// TwinCAT 3 PLC project Project_02
// ProgramVersion: 3.1.4024.0
// libraries:
//   Tc2_Standard, * (Beckhoff Automation GmbH)
//   Tc2_System, * (Beckhoff Automation GmbH)
//   Tc3_Module, * (Beckhoff Automation GmbH)
// project tree:
//   DUTs/ DUT.TcTLEO
//   GVLs/ InputOutput.TcGVL
//   / PlcTask.TcTTO
//   POUs/ FB_MSF.TcPOU, FB_oscillatore.TcPOU, MAIN.TcPOU

CONFIGURATION Project_02
    RESOURCE PLC ON TwinCAT3
        TASK PlcTask(INTERVAL := T#10ms, PRIORITY := 20);
        PROGRAM MAIN WITH PlcTask : MAIN;
    END_RESOURCE
END_CONFIGURATION

// ---- DUTs/DUT.TcTLEO
{attribute 'qualified_only'}
{attribute 'strict'}

TYPE STATI :
(
	S0 := 0, S1, S2, S3, SE, SA
);
END_TYPE

// ---- GVLs/InputOutput.TcGVL
{attribute 'qualified_only'}
VAR_GLOBAL
	start  : BOOL;
	stop   : BOOL;
	emg    : BOOL;
	ack    : BOOL;
	fc1    : BOOL;
	fc2    : BOOL;
	
	H1     : BOOL;
	HEMG   : BOOL;
	M      : BOOL;
	libero : BOOL;
	
END_VAR

// ---- POUs/MAIN.TcPOU
PROGRAM MAIN
VAR
	nastro: FB_MSF();
	emg: BOOL;
END_VAR


nastro(
	start:= InputOutput.start, 
	stop:= InputOutput.stop, 
	emg:= InputOutput.emg, 
	ack:= InputOutput.ack, 
	fc1:= InputOutput.fc1, 
	fc2:= InputOutput.fc2, 
	H1=> InputOutput.H1, 
	HEMG=> InputOutput.HEMG, 
	M=> InputOutput.M, 
	libero=> InputOutput.libero);

END_PROGRAM

// ---- POUs/FB_MSF.TcPOU
FUNCTION_BLOCK FB_MSF
VAR_INPUT
	start: BOOL;
	stop : BOOL := TRUE;
	emg  : BOOL := TRUE;
	ack  : BOOL;
	fc1  : BOOL;
	fc2  : BOOL;
END_VAR
VAR_OUTPUT
	H1   : BOOL;
	HEMG : BOOL;
	M    : BOOL;
	// il nastro è libero
	libero : BOOL;
END_VAR
VAR
	
	// abilitazione dell’automatismo
	enable : BOOL := TRUE;
	// condizioni di transizione
	tr_S0_S1 : BOOL;
	tr_S1_S2 : BOOL;
	tr_S2_S3 : BOOL;
	tr_S3_S1 : BOOL;
	tr_S3_S0 : BOOL;
	tr_SE_SA : BOOL;
	tr_SA_S0 : BOOL;
	// variabile di stato
	stato : STATI := STATI.S0;
	// timers
	T31 : TON();
	TA0 : TON();
	// triggers per segnalazione nastro libero
	pckin : R_TRIG();
	pckout: R_TRIG();
	// lampeggio
	osc : FB_oscillatore();	
END_VAR

(*
1.aggiornamento delle condizioni di abilitazione (stop, allarmi, etc)
2.aggiornamento di timers, contatori, triggers sui fronti
3.valutazione della condizione di arresto nominale
4.valutazione della condizione di arresto di emergenza
5.aggiornamento delle condizioni di transizione di stato
6.switch-case della MSF
7.comando delle uscite
*)
// 1. aggiornamento condizioni di abilitazione
enable := stop AND emg;
// 2. aggiornamento timers, contatori, triggers sui fronti
T31(IN := (stato = STATI.S3 AND enable), PT := T#10S);
TA0(IN := (stato = STATI.SA AND enable), PT := T#10S);
pckin(clk:= fc1);
pckout(clk:= fc2);
osc(enable := (stato = STATI.SA), t_high := T#500MS, t_low := T#500MS);

// 3. condizione di arresto nominale
IF NOT stop AND emg THEN
	stato := STATI.S0;	
END_IF
// 4. condizione di arresto di emergenza
IF NOT emg THEN
	stato := STATI.SE;
END_IF
// 5. aggiornamento delle condizioni di transizione
tr_S0_S1 := enable AND start;
tr_S1_S2 := enable AND fc1 AND NOT fc2;
tr_S2_S3 := enable AND fc2;
tr_S3_S1 := enable AND fc1 AND NOT fc2 AND NOT T31.Q;
tr_S3_S0 := enable AND T31.Q;
tr_SE_SA := enable AND ack;
tr_SA_S0 := enable AND TA0.Q;
// 6. switch-case della MSF
CASE stato OF
STATI.S0:
	IF tr_S0_S1 THEN
		stato := STATI.S1;
	END_IF
STATI.S1:
	IF tr_S1_S2 THEN
		stato := STATI.S2;
	END_IF
STATI.S2:
	IF tr_S2_S3 THEN
		stato := STATI.S3;
	END_IF
STATI.S3:
	IF tr_S3_S1 THEN
		stato := STATI.S1;
	ELSIF tr_S3_S0 THEN
		stato := STATI.S0;
	END_IF
STATI.SE:
	IF tr_SE_SA THEN
		stato := STATI.SA;
	END_IF
STATI.SA:
	IF tr_SA_S0 THEN
		stato := STATI.S0;
	END_IF
ELSE
	stato := STATI.SE;
END_CASE
// 7. comando uscite
H1 := stato <> STATI.S0;
HEMG := (stato = STATI.SE) OR osc.q;
M := (stato = STATI.S2) OR (stato = STATI.S3);
// nastro libero se (enable = true e  pckout.q) o (fc1 libero in S1);
// nastro occupato se enable = false o fc1.rise o stato = S0
IF (enable AND (pckout.q)) OR (stato = STATI.S1 AND NOT fc1) THEN
	libero := TRUE;
ELSIF (NOT enable) OR pckin.Q OR stato = STATI.S0 THEN
	libero := FALSE;
END_IF

END_FUNCTION_BLOCK

// ---- POUs/FB_oscillatore.TcPOU
FUNCTION_BLOCK FB_oscillatore
VAR_INPUT
	enable   : BOOL;
	t_high   : TIME;
	t_low    : TIME;
END_VAR
VAR_OUTPUT
	q        : BOOL;
END_VAR
VAR
    t1       : TON();
	t2       : TON();
END_VAR

t1(in := enable AND NOT t2.Q, pt := t_low);
t2(in := t1.Q, pt := t_high);

q := t1.Q;

END_FUNCTION_BLOCK
